(* Schneider Machine Expert - Basic project Kali bagi tambah kurang, file version 1.7.0.0 *)
(* ProjectInformations: Name=New project *)

HARDWARE
  Cpu 0: TM221ME32TK
  EthernetConfiguration: NetworkName=M221, IpAllocationMode=FixedAddress, IpAddress=0.0.0.0, SubnetMask=0.0.0.0
  SerialLineConfiguration: Baud=Baud19200, Parity=ParityEven, DataBits=DataBits8, StopBits=StopBits1, PhysicalMedium=PhysicalMediumRs485, TransmissionMode=TransmissionModeModbusRtu, SlaveId=1, Addressing=SlaveAddressing
  MastTask: UsePeriodScanMode=false, PeriodScan=100
  FastTask: Period=255
  CpuBehavior: StartingMode=StartAsPreviousState, AutoSaveRamOnEeprom=true, WatchdogPeriod=250

SYMBOLS  (address, symbol, comment, settings)

POU New POU
  (* SectionNumber=1 *)

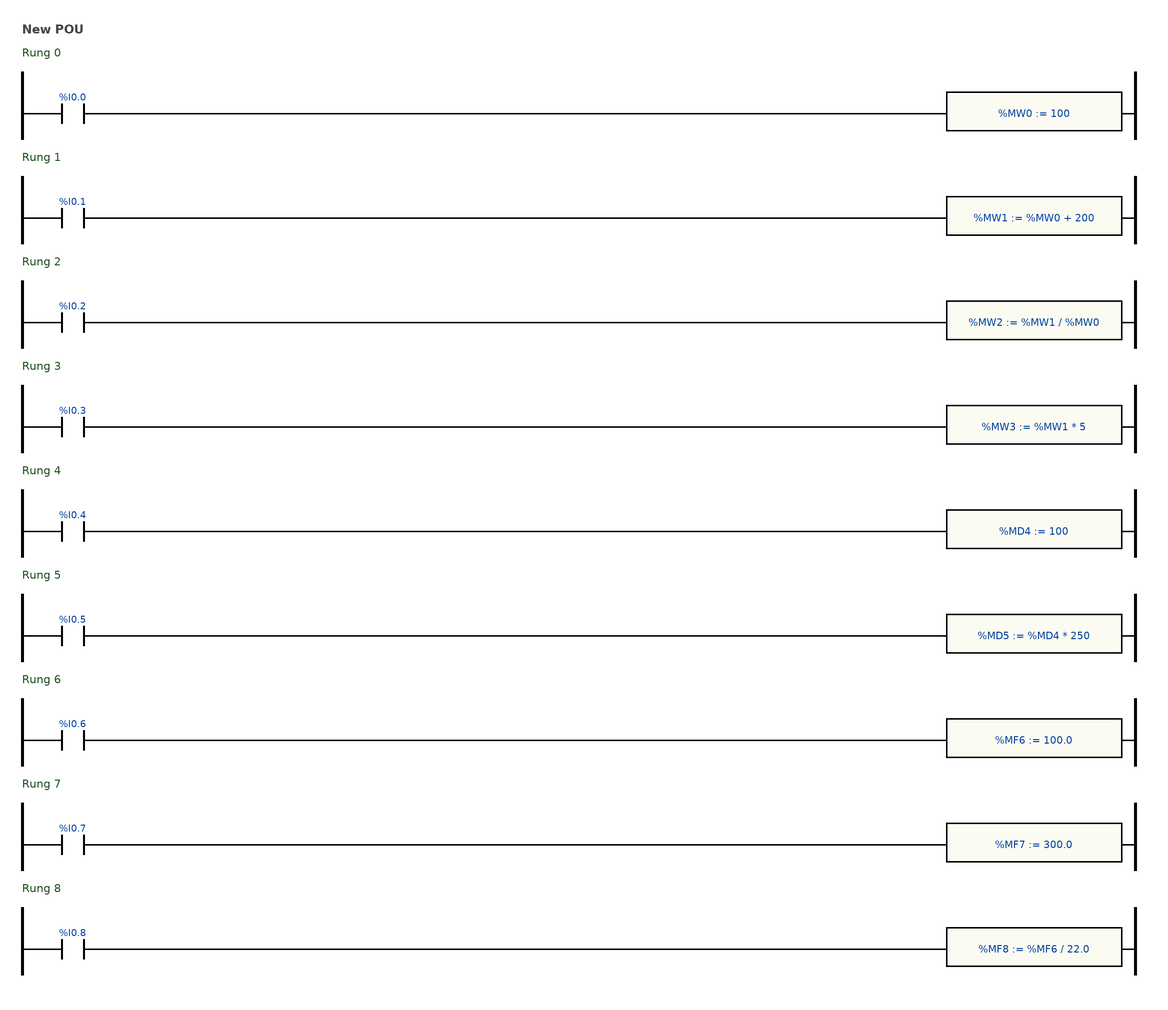

// Rung 0
  LD %I0.0
  [ %MW0 := 100 ]
  // as ST:
  //   IF %I0.0 THEN %MW0 := 100; END_IF;

// Rung 1
  LD %I0.1
  [ %MW1 := %MW0 + 200 ]
  // as ST:
  //   IF %I0.1 THEN %MW1 := %MW0 + 200; END_IF;

// Rung 2
  LD %I0.2
  [ %MW2 := %MW1 / %MW0 ]
  // as ST:
  //   IF %I0.2 THEN %MW2 := %MW1 / %MW0; END_IF;

// Rung 3
  LD %I0.3
  [ %MW3 := %MW1 * 5 ]
  // as ST:
  //   IF %I0.3 THEN %MW3 := %MW1 * 5; END_IF;

// Rung 4
  LD %I0.4
  [ %MD4 := 100 ]
  // as ST:
  //   IF %I0.4 THEN %MD4 := 100; END_IF;

// Rung 5
  LD %I0.5
  [ %MD5 := %MD4 * 250 ]
  // as ST:
  //   IF %I0.5 THEN %MD5 := %MD4 * 250; END_IF;

// Rung 6
  LD %I0.6
  [ %MF6 := 100.0 ]
  // as ST:
  //   IF %I0.6 THEN %MF6 := 100.0; END_IF;

// Rung 7
  LD %I0.7
  [ %MF7 := 300.0 ]
  // as ST:
  //   IF %I0.7 THEN %MF7 := 300.0; END_IF;

// Rung 8
  LD %I0.8
  [ %MF8 := %MF6 / 22.0 ]
  // as ST:
  //   IF %I0.8 THEN %MF8 := %MF6  /  22.0; END_IF;
